FUNCTION_BLOCK Palletizer EXTENDS A_Actuator
VAR_INPUT
	fbBeltConveyor : Conveyor;
	fbPalletizerChain : Conveyor;
	fbRollerConveyor : Conveyor;
	fbTurnCylinder : Cylinder;
	fbClamperCylinder : Cylinder;
	fbPusherCylinder : Cylinder;
	fbPlateCylinder : Cylinder;
	fbElevator : Elevator; 
END_VAR
VAR_OUTPUT
	
END_VAR
VAR

END_VAR

METHOD  executeCmd : BOOL
VAR_INPUT
	
END_VAR
END_METHOD

END_FUNCTION_BLOCK

(* stored: Version 1.1.0.1, ProductVersion 3.1.4024.2
   POU Palletizer: Id {bec17fcd-d370-4629-83c7-5c1536ecde34}, SpecialFunc None
   Method executeCmd: Id {662cb160-8947-48d0-b2fc-2803db90e6e7} *)
